// TIA Portal V19 export
TYPE "LAF_typeConstraintRollerEm2ParametersInterfaceHmi"
// stored: Access Published
   STRUCT
      configuration : "LAF_typeConstraintRollerEm2ParametersHmi";
      commands : "LBC_typeInterfaceCommands";
      monitoring { S7_SetPoint := 'True'} : "LAF_typeConstraintRollerEm2ProcessValuesHmi";
   END_STRUCT;
END_TYPE
